// TIA Portal V17 export
// export: Created 2025-04-09T07:53:26.6449027Z, ExportSetting WithDefaults, DisplayName Totally Integrated Automation Portal, DisplayVersion V17, DisplayName TIA Portal Openness, DisplayVersion V17, DisplayName TIA Portal Version Control Interface, DisplayVersion V17, DisplayName STEP 7 Professional, DisplayVersion V17, DisplayName STEP 7 Safety, DisplayVersion V17, DisplayName WinCC Advanced, DisplayVersion V17
TYPE "User_data_type_1"
// stored: IsFailsafeCompliant false
   STRUCT
      Input : AOM_IDENT;
   END_STRUCT;
END_TYPE
